// TwinCAT 3 PLC project test
// ProgramVersion: 3.1.4026.17
// libraries:
//   Tc2_Standard, * (Beckhoff Automation GmbH)
//   Tc2_System, * (Beckhoff Automation GmbH)
//   Tc2_Utilities, * (Beckhoff Automation GmbH)
// project tree:
//   Lib/CircularFifoBuffer/ CircularFifoBuffer.TcPOU
//   Lib/ReadersWriters/Base/ Reader.TcIO, Writer.TcIO
//   Lib/ReadersWriters/Buffered/ BufferedReader.TcPOU, BufferedWriter.TcPOU
//   Lib/Streams/ InputStream.TcIO, OutputStream.TcIO
//   Programs/ Test.TcPOU
//   Tasks/ PlcTask.TcTTO
// real-time tasks:
//   TASK PlcTask: cycle T#10ms, priority 20, ADS port 350

CONFIGURATION test
    RESOURCE PLC ON TwinCAT3
        TASK PlcTask(INTERVAL := T#10ms, PRIORITY := 20);
        PROGRAM Test WITH PlcTask : Test;
    END_RESOURCE
END_CONFIGURATION

// ---- Lib/ReadersWriters/Base/Reader.TcIO
INTERFACE PUBLIC Reader EXTENDS __SYSTEM.IQueryInterface

END_INTERFACE

// ---- Lib/ReadersWriters/Base/Writer.TcIO
INTERFACE PUBLIC Writer EXTENDS __SYSTEM.IQueryInterface

END_INTERFACE

// ---- Lib/Streams/InputStream.TcIO
INTERFACE PUBLIC InputStream EXTENDS __SYSTEM.IQueryInterface

PROPERTY PUBLIC Available : UDINT
GET
END_GET
END_PROPERTY

PROPERTY PUBLIC IsMarkSupported : BOOL
GET
END_GET
END_PROPERTY

METHOD PUBLIC Mark
VAR_INPUT
	read_limit : UDINT;
END_VAR
END_METHOD

METHOD Read : BOOL
VAR_OUTPUT
	data : BYTE;
END_VAR
END_METHOD

METHOD ReadByteArray : BOOL
VAR_OUTPUT
	data_pointer : POINTER TO BYTE;
	len : UDINT;
END_VAR
END_METHOD

METHOD PUBLIC Reset
END_METHOD

METHOD Skip : UDINT
VAR_INPUT
	n : UDINT;
END_VAR
END_METHOD

END_INTERFACE

// ---- Lib/Streams/OutputStream.TcIO
INTERFACE PUBLIC OutputStream EXTENDS __System.IQueryInterface

METHOD PUBLIC Close
END_METHOD

METHOD PUBLIC Flush
END_METHOD

METHOD Write : BOOL
VAR_INPUT
	data : BYTE;
END_VAR
END_METHOD

METHOD WriteByteArray : BOOL
VAR_INPUT
	data_pointer : POINTER TO BYTE;
	len : UDINT;
END_VAR
END_METHOD

END_INTERFACE

// ---- Programs/Test.TcPOU
PROGRAM Test
VAR
	cfb : CircularFifoBuffer<256>;
	reader : BufferedReader(input_stream := cfb);
	string_to_write : T_MaxString := 'Start';
	bytes_to_write : ARRAY[0..MAX_STRING_LENGTH] OF BYTE;
	
	write : BOOL;	
	write_partial : BOOL;
	write_line_end : BOOL;
	
	received_line : T_MaxString;
	
	{attribute 'hide'} temp_line : T_MaxString;	
	{attribute 'hide'} i : INT;
END_VAR

IF write THEN
	write := FALSE;
	IF INT_TO_UDINT(LEN(string_to_write)) < cfb.SpaceLeft THEN
		bytes_to_write := MAXSTRING_TO_BYTEARR(string_to_write);
		
		FOR i := 0 TO LEN(string_to_write) DO
			cfb.Write(bytes_to_write[i]);
		END_FOR
	END_IF
END_IF

IF write_partial THEN
	write_partial := FALSE;
	IF INT_TO_UDINT(LEN(string_to_write)) < cfb.SpaceLeft THEN
		bytes_to_write := MAXSTRING_TO_BYTEARR(string_to_write);
		
		FOR i := 0 TO LEN(string_to_write) - 1 DO
			cfb.Write(bytes_to_write[i]);
		END_FOR
	END_IF
END_IF

IF write_line_end THEN
	write_line_end := FALSE;
	
	IF cfb.SpaceLeft > 0 THEN
		cfb.Write(0);
	END_IF
END_IF

IF reader.ReadLine(line => temp_line) THEN
	received_line := temp_line;
END_IF

END_PROGRAM

// ---- Lib/CircularFifoBuffer/CircularFifoBuffer.TcPOU
{attribute 'linkalways'} 
{attribute 'no_explicit_call' := 'This FB is a CLASS and must be accessed using methods or properties'}
{attribute 'enable_dynamic_creation'}
FUNCTION_BLOCK PUBLIC CircularFifoBuffer
VAR_GENERIC CONSTANT
	capacity : UDINT := 64;
END_VAR
IMPLEMENTS InputStream, OutputStream
VAR
	buffer : ARRAY[0..capacity-1] OF BYTE;
	read_position : UDINT;
	write_position : UDINT;
	mark_position : UDINT;
	mark_size : UDINT;
END_VAR

{attribute 'monitoring' := 'call'}
PROPERTY PUBLIC Available : UDINT
GET // PUBLIC
IF read_position <= write_position THEN
	// any space between the first read and
	// the first write is available.  In this case i
	// is all in one piece.
	Available := write_position - read_position;
	RETURN;
END_IF

// space at the beginning and end.
Available := capacity - (read_position - write_Position);
END_GET
END_PROPERTY

METHOD PUBLIC Clear
read_position := 0;
write_position := 0;
mark_position := 0;
END_METHOD

{warning 'Add method implementation '}
METHOD PUBLIC Close
END_METHOD

METHOD INTERNAL EnsureMark
IF Marked > mark_size THEN
	mark_position := read_position;
	mark_size := 0;
END_IF
END_METHOD

{warning 'Add method implementation '}
METHOD PUBLIC Flush
END_METHOD

{attribute 'monitoring' := 'call'}
PROPERTY PUBLIC IsMarkSupported : BOOL
GET // PUBLIC
IsMarkSupported := FALSE;
END_GET
END_PROPERTY

METHOD PUBLIC Mark
VAR_INPUT
	read_limit : UDINT;
END_VAR
END_METHOD

{attribute 'monitoring' := 'call'}
PROPERTY PUBLIC Marked : UDINT
GET // PUBLIC
IF mark_position <= read_position THEN
	// any space between the markPosition and
	// the first write is marked.  In this case i
	// is all in one piece.
	Marked := read_position - mark_position;
	RETURN;
END_IF

// space at the beginning and end.
Marked := capacity - (mark_position - read_position);
END_GET
END_PROPERTY

METHOD PUBLIC Read : BOOL
VAR_OUTPUT
	data : BYTE;
END_VAR
IF Available > 0 THEN
	data := buffer[read_position];
	read_position := read_position + 1;
	Read := TRUE;
	
	IF read_position = capacity THEN
		read_position := 0;
	END_IF
	
	EnsureMark();
END_IF
END_METHOD

{warning 'Add method implementation '}
METHOD PUBLIC ReadByteArray : BOOL
VAR_OUTPUT
	data_pointer : POINTER TO BYTE;
	len : UDINT;
END_VAR
END_METHOD

METHOD PUBLIC Reset
END_METHOD

{attribute 'monitoring' := 'call'}
PROPERTY PUBLIC Size : UDINT
GET // PUBLIC
Size := capacity;
END_GET
END_PROPERTY

METHOD PUBLIC Skip : UDINT
VAR_INPUT
	n : UDINT;
END_VAR
END_METHOD

{attribute 'monitoring' := 'call'}
PROPERTY PUBLIC SpaceLeft : UDINT
GET // PUBLIC
IF write_position < mark_position THEN
	// any space between the first write and
	// the mark except one byte is available.
	// In this case it is all in one piece.
	SpaceLeft := mark_position - write_position - 1;
	RETURN;
END_IF

// space at the beginning and end.
SpaceLeft := (capacity - 1) - (write_position - mark_position);
END_GET
END_PROPERTY

METHOD PUBLIC Write : BOOL
VAR_INPUT
	data : BYTE;
END_VAR
IF SpaceLeft < 1 THEN
	RETURN;
END_IF

buffer[write_position] := data;

write_position := write_position + 1;

IF write_position = capacity THEN
	write_position := 0;
END_IF

Write := TRUE;
END_METHOD

METHOD PUBLIC WriteByteArray : BOOL
VAR_INPUT
	data_pointer : POINTER TO BYTE;
	len : UDINT;
END_VAR
VAR
	i : UDINT;
	ptr : POINTER TO BYTE;
END_VAR
IF len <= SpaceLeft THEN
	FOR i := 0 TO len DO
		ptr := data_pointer + 1;
		IF NOT Write(ptr^) THEN
			RETURN;
		END_IF
	END_FOR
END_IF
END_METHOD

END_FUNCTION_BLOCK

// ---- Lib/ReadersWriters/Buffered/BufferedReader.TcPOU
{attribute 'linkalways'} 
{attribute 'no_explicit_call' := 'This FB is a CLASS and must be accessed using methods or properties'}
{attribute 'enable_dynamic_creation'}
FUNCTION_BLOCK BufferedReader IMPLEMENTS Reader
VAR
	input_stream : InputStream;
END_VAR

//FB_Init is always available implicitly and it is used primarily for initialization.
//The return value is not evaluated. For a specific influence, you can also declare the
//methods explicitly and provide additional code there with the standard initialization
//code. You can evaluate the return value.
METHOD FB_Init: BOOL
VAR_INPUT
    bInitRetains: BOOL; // TRUE: the retain variables are initialized (reset warm / reset cold)
    bInCopyCode: BOOL;  // TRUE: the instance will be copied to the copy code afterward (online change)
	input_stream : InputStream;
END_VAR
THIS^.input_stream := input_stream;
END_METHOD

METHOD PUBLIC ReadLine : BOOL
VAR_OUTPUT
	line : T_MaxString;
END_VAR
VAR_INST
	i : INT;
	data : ARRAY[0..MAX_STRING_LENGTH] OF BYTE;
END_VAR
VAR
	read_byte : BYTE;
END_VAR
IF input_stream.Read(data => read_byte) THEN
	data[i] := read_byte;
	IF data[i] = 0 THEN
		line := BYTEARR_TO_MAXSTRING(data);
		ReadLine := TRUE;
		i := 0;
	ELSE
		i := i + 1;
	END_IF
END_IF
END_METHOD

END_FUNCTION_BLOCK

// ---- Lib/ReadersWriters/Buffered/BufferedWriter.TcPOU
{attribute 'linkalways'} 
{attribute 'no_explicit_call' := 'This FB is a CLASS and must be accessed using methods or properties'}
{attribute 'enable_dynamic_creation'}
FUNCTION_BLOCK BufferedWriter IMPLEMENTS Writer
VAR
	output_stream : OutputStream;
END_VAR

//FB_Init is always available implicitly and it is used primarily for initialization.
//The return value is not evaluated. For a specific influence, you can also declare the
//methods explicitly and provide additional code there with the standard initialization
//code. You can evaluate the return value.
METHOD FB_Init: BOOL
VAR_INPUT
    bInitRetains: BOOL; // TRUE: the retain variables are initialized (reset warm / reset cold)
    bInCopyCode: BOOL;  // TRUE: the instance will be copied to the copy code afterward (online change)
	output_stream : OutputStream;
END_VAR
THIS^.output_stream := output_stream;
END_METHOD

METHOD PUBLIC WriteLine : BOOL
VAR_INPUT
	line : T_MaxString;
END_VAR
END_METHOD

END_FUNCTION_BLOCK
